Staubli VAL3: onSpaceEvent.pgx

program onSpaceEvent(string x_sId)
  local bool l_bStatus
  local num l_nX
  local num l_nValue
  local string l_sString
  local num l_nY
  local bool l_bOk
begin
  //
  // NB sEvent is the selected
  // element in the LIST
  //
  //
  if nViewMode==0
    call out:getStatus(l_bStatus,x_sId)
    call out:setStatus(!l_bStatus,x_sId)
    logMsg("[KERNEL] INTERFACE:Change the status ON/OFF of: "+sEvent)
  elseIf nViewMode==2
    if find(x_sId,"In")!=-1
      // INPUT not allowed
      return
    else
      l_nX=40-use:nBottomX+find(sEvent,"[")
      call saveInOut:getValue_num(l_nValue,x_sId)
      l_sString=toString("3",l_nValue)
    endIf
    // set IT
    l_nY=nView+1
    call use:read(l_nX,l_nY,l_sString,14,false)
    // COUNT
    toNum(l_sString,l_nValue,l_bOk)
    if l_bOk
      // set the value
      call NUM:setValue(l_nValue,x_sId)
    endIf
  endIf
end
